FUNCTION_BLOCK Label 
VAR
	_label : T_MaxString;
END_VAR

PROPERTY Text : STRING
GET
Text := _label;
END_GET
SET
_label := Text;
END_SET
END_PROPERTY

END_FUNCTION_BLOCK

(* stored: Version 1.1.0.1, ProductVersion 3.1.4024.12
   POU Label: Id {407f426c-0c4c-4de9-b8b0-502b37790a3f}, SpecialFunc None
   Property Text: Id {66237e83-5a30-47d6-bcb8-5508ec49c1c4}
   Get Get: Id {dc89a7b6-455a-4823-a351-6300d9e79d42}
   Set Set: Id {a47bba9f-441b-4460-8539-be58aceacbb1} *)
